FUNCTION "SM_GetState" : Int
{ S7_Optimized_Access := 'FALSE' }
VERSION : 0.1
   VAR_IN_OUT
      inst : "typeSM";
   END_VAR


BEGIN
	#SM_GetState := #inst.state;
END_FUNCTION

